TYPE ST_Setup_ECS :
STRUCT
	bOnEmergPowerOff				: BOOL;				//When emergency power is active then user can choose if the device is on or switch automatic off
	bManualyOn						: BOOL;				//Switch the device manualy on
	byPriority						: BYTE; 			//{#lynus.ag#()} //Priority of the device if controlled via the EMS block = 1 2 3 (If 0 then this device does not exist for the EMS block)
	byEnableSOC						: BYTE; 			//{#lynus.ag#()} //Enable the device when the battery SOC is greater than equal this value
	byDisableSOC					: BYTE; 			//{#lynus.ag#()} //Disable the device when the battery SOC is smaler than equal this value
	byManualyTargetPower			: BYTE;				//% of the max Power in kW when the Device is manually on
	byCSMinPower					: BYTE;				//{#lynus.ag#()} //Min power in % of the max power in kW. The charging station is operated with this power even if there is no surplus.
	rMaxPower						: REAL; 			//{#lynus.ag#()} //Max. power from the charging Station with unit kW
END_STRUCT
END_TYPE

(* stored: Version 1.1.0.1, ProductVersion 3.1.4024.6
   DUT ST_Setup_ECS: Id {9f07984e-39c4-42a1-9d12-fedfd4ffc38a} *)
